FUNCTION_BLOCK RT_E_TRAIN (* Generation of a finite train of events *)
  (* Standard: 61499-2 *)
  (* Version 0.0, 2008-07-10, 4DIAC-IDE, 4DIAC-Consortium *)
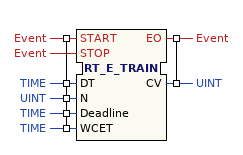
  EVENT_INPUT
    START WITH DT, N, Deadline, WCET;
    STOP;
  END_EVENT
  EVENT_OUTPUT
    EO WITH CV; (* N events at period DT,starting at DT after START *)
  END_EVENT
  VAR_INPUT
    DT : TIME; (* Period between events *)
    N : UINT; (* Number of events to generate *)
    Deadline : TIME;
    WCET : TIME;
  END_VAR
  VAR_OUTPUT
    CV : UINT; (* EO index(0 N-1) *)
  END_VAR
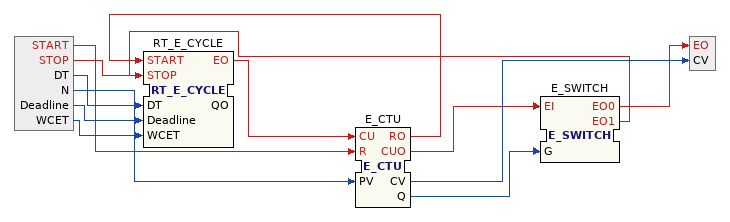
  FBS
    RT_E_CYCLE : RT_E_CYCLE;
    E_CTU : E_CTU;
    E_SWITCH : E_SWITCH;
  END_FBS
  EVENT_CONNECTIONS
    RT_E_CYCLE.EO TO E_CTU.CU;
    START TO E_CTU.R;
    STOP TO RT_E_CYCLE.STOP;
    E_CTU.RO TO RT_E_CYCLE.START;
    E_CTU.CUO TO E_SWITCH.EI;
    E_SWITCH.EO0 TO EO;
    E_SWITCH.EO1 TO RT_E_CYCLE.STOP;
  END_CONNECTIONS
  DATA_CONNECTIONS
    DT TO RT_E_CYCLE.DT;
    Deadline TO RT_E_CYCLE.Deadline;
    WCET TO RT_E_CYCLE.WCET;
    N TO E_CTU.PV;
    E_CTU.CV TO CV;
    E_CTU.Q TO E_SWITCH.G;
  END_CONNECTIONS
END_FUNCTION_BLOCK
